FUNCTION_BLOCK Timer
VAR_INPUT
	EN: BOOL := TRUE;
END_VAR
VAR_OUTPUT
	ET: LTIME;
END_VAR
VAR
    _TimeTick: LINT;
    _StartTick: LINT;
    _Timeout: BOOL;
END_VAR

ET := LINT_TO_LTIME(ElapsedTime() * 1000000);
IF NOT EN THEN
	Restart();
END_IF

METHOD ElapsedTime : LINT
VAR_INPUT
END_VAR
IF EN THEN
	ElapsedTime := (GetTickCount() - _StartTick);
ELSE
	ElapsedTime := 0;	
END_IF
END_METHOD

METHOD FB_init : BOOL
VAR_INPUT
	bInitRetains : BOOL; // if TRUE, the retain variables are initialized (warm start / cold start)
	bInCopyCode : BOOL;  // if TRUE, the instance afterwards gets moved into the copy code (online change)
END_VAR
TimeoutTime := 1000;
Restart();
END_METHOD

METHOD Restart : BOOL
VAR_INPUT
END_VAR
_Timeout := FALSE;
_StartTick := GetTickCount();
Restart := TRUE;
END_METHOD

METHOD Timeout : BOOL
VAR_INPUT
END_VAR
IF NOT _Timeout THEN
	IF (GetTickCount() - _StartTick) >= _TimeTick THEN
		_Timeout := TRUE;
	END_IF
END_IF
Timeout := _Timeout;
END_METHOD

PROPERTY TimeoutTime : LINT
GET
TimeoutTime := _TimeTick;
END_GET
SET
VAR
	Temp: lint;
END_VAR
Temp := TimeoutTime;
IF (TimeoutTime > 0) AND (Temp <= 1) THEN
	Temp := 2; { Smallest timeout }
END_IF
IF Temp <> _TimeTick THEN
	_TimeTick := Temp;
	Restart();
END_IF
END_SET
END_PROPERTY

END_FUNCTION_BLOCK

(* stored: Version 1.1.0.1, ProductVersion 3.1.4024.4
   POU Timer: Id {7e40e161-4977-4818-ba36-1d51bb135bda}, SpecialFunc None
   Method ElapsedTime: Id {4e685e91-bd49-4516-b927-236d0d0f0eaa}
   Method FB_init: Id {119615cf-dd7a-423d-95a6-7ed2302d12e3}
   Method Restart: Id {d54a3879-94a5-49f6-bcde-47b508c56933}
   Method Timeout: Id {15717f88-1ef3-438f-83ed-d1058b2fb2bc}
   Property TimeoutTime: Id {61ed3f75-0994-47ab-9a94-064aeb46ab2e}
   Get Get: Id {d6646e3c-e277-45da-a165-a0e9a4e8d2f7}
   Set Set: Id {020752f4-0484-4707-ac32-7e259f5a1f32} *)
